// TIA Portal V19 export
FUNCTION "AUTO_SUBOUTPUT" : Void   // FC9, LAD
{ S7_Optimized_Access := 'TRUE' }
// stored: SetENOAutomatically false
BEGIN

REGION Network 1: P-202 A RO 1 FEED PUMP
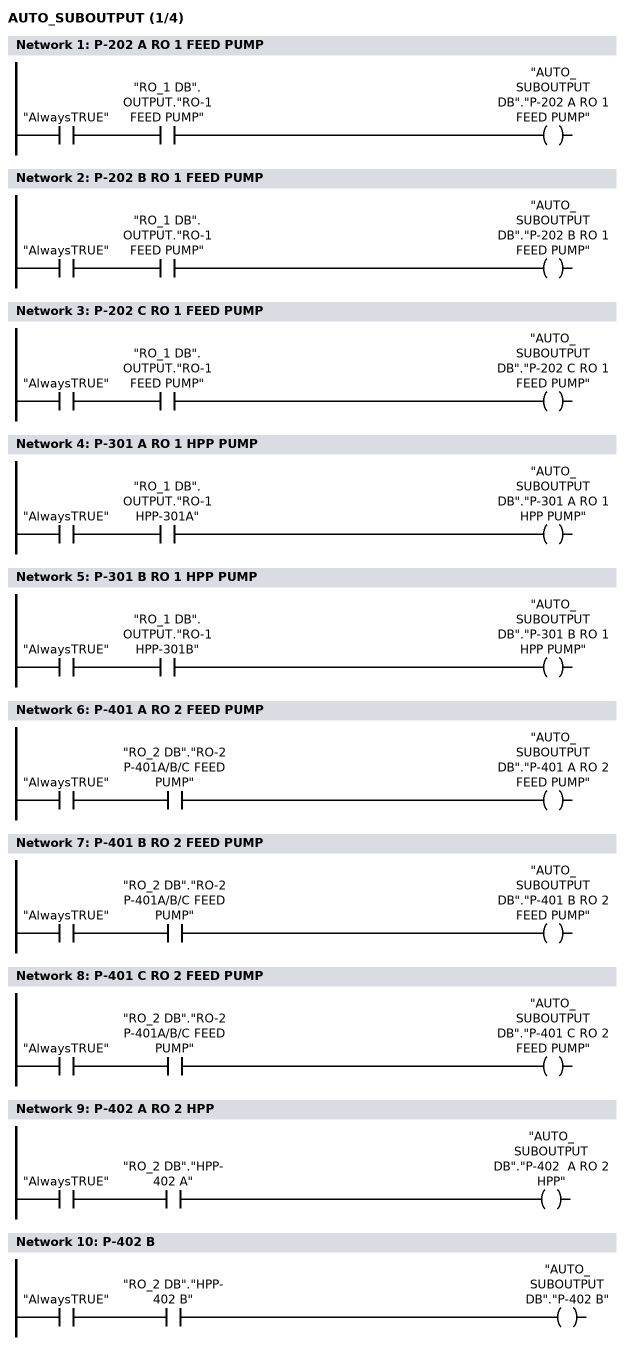
   RUNG wire#powerrail
      Contact( "AlwaysTRUE" )
      Contact( "RO_1 DB".OUTPUT."RO-1 FEED PUMP" )
      Coil( "AUTO_SUBOUTPUT DB"."P-202 A RO 1 FEED PUMP" )
   END_RUNG
   // the same network as SCL:
   "AUTO_SUBOUTPUT DB"."P-202 A RO 1 FEED PUMP" := "AlwaysTRUE" AND "RO_1 DB".OUTPUT."RO-1 FEED PUMP";
END_REGION

REGION Network 2: P-202 B RO 1 FEED PUMP
   RUNG wire#powerrail
      Contact( "AlwaysTRUE" )
      Contact( "RO_1 DB".OUTPUT."RO-1 FEED PUMP" )
      Coil( "AUTO_SUBOUTPUT DB"."P-202 B RO 1 FEED PUMP" )
   END_RUNG
   // the same network as SCL:
   "AUTO_SUBOUTPUT DB"."P-202 B RO 1 FEED PUMP" := "AlwaysTRUE" AND "RO_1 DB".OUTPUT."RO-1 FEED PUMP";
END_REGION

REGION Network 3: P-202 C RO 1 FEED PUMP
   RUNG wire#powerrail
      Contact( "AlwaysTRUE" )
      Contact( "RO_1 DB".OUTPUT."RO-1 FEED PUMP" )
      Coil( "AUTO_SUBOUTPUT DB"."P-202 C RO 1 FEED PUMP" )
   END_RUNG
   // the same network as SCL:
   "AUTO_SUBOUTPUT DB"."P-202 C RO 1 FEED PUMP" := "AlwaysTRUE" AND "RO_1 DB".OUTPUT."RO-1 FEED PUMP";
END_REGION

REGION Network 4: P-301 A RO 1 HPP PUMP
   RUNG wire#powerrail
      Contact( "AlwaysTRUE" )
      Contact( "RO_1 DB".OUTPUT."RO-1 HPP-301A" )
      Coil( "AUTO_SUBOUTPUT DB"."P-301 A RO 1 HPP PUMP" )
   END_RUNG
   // the same network as SCL:
   "AUTO_SUBOUTPUT DB"."P-301 A RO 1 HPP PUMP" := "AlwaysTRUE" AND "RO_1 DB".OUTPUT."RO-1 HPP-301A";
END_REGION

REGION Network 5: P-301 B RO 1 HPP PUMP
   RUNG wire#powerrail
      Contact( "AlwaysTRUE" )
      Contact( "RO_1 DB".OUTPUT."RO-1 HPP-301B" )
      Coil( "AUTO_SUBOUTPUT DB"."P-301 B RO 1 HPP PUMP" )
   END_RUNG
   // the same network as SCL:
   "AUTO_SUBOUTPUT DB"."P-301 B RO 1 HPP PUMP" := "AlwaysTRUE" AND "RO_1 DB".OUTPUT."RO-1 HPP-301B";
END_REGION

REGION Network 6: P-401 A RO 2 FEED PUMP
   RUNG wire#powerrail
      Contact( "AlwaysTRUE" )
      Contact( "RO_2 DB"."RO-2 P-401A/B/C FEED PUMP" )
      Coil( "AUTO_SUBOUTPUT DB"."P-401 A RO 2 FEED PUMP" )
   END_RUNG
   // the same network as SCL:
   "AUTO_SUBOUTPUT DB"."P-401 A RO 2 FEED PUMP" := "AlwaysTRUE" AND "RO_2 DB"."RO-2 P-401A/B/C FEED PUMP";
END_REGION

REGION Network 7: P-401 B RO 2 FEED PUMP
   RUNG wire#powerrail
      Contact( "AlwaysTRUE" )
      Contact( "RO_2 DB"."RO-2 P-401A/B/C FEED PUMP" )
      Coil( "AUTO_SUBOUTPUT DB"."P-401 B RO 2 FEED PUMP" )
   END_RUNG
   // the same network as SCL:
   "AUTO_SUBOUTPUT DB"."P-401 B RO 2 FEED PUMP" := "AlwaysTRUE" AND "RO_2 DB"."RO-2 P-401A/B/C FEED PUMP";
END_REGION

REGION Network 8: P-401 C RO 2 FEED PUMP
   RUNG wire#powerrail
      Contact( "AlwaysTRUE" )
      Contact( "RO_2 DB"."RO-2 P-401A/B/C FEED PUMP" )
      Coil( "AUTO_SUBOUTPUT DB"."P-401 C RO 2 FEED PUMP" )
   END_RUNG
   // the same network as SCL:
   "AUTO_SUBOUTPUT DB"."P-401 C RO 2 FEED PUMP" := "AlwaysTRUE" AND "RO_2 DB"."RO-2 P-401A/B/C FEED PUMP";
END_REGION

REGION Network 9: P-402 A RO 2 HPP
   RUNG wire#powerrail
      Contact( "AlwaysTRUE" )
      Contact( "RO_2 DB"."HPP-402 A" )
      Coil( "AUTO_SUBOUTPUT DB"."P-402  A RO 2 HPP" )
   END_RUNG
   // the same network as SCL:
   "AUTO_SUBOUTPUT DB"."P-402  A RO 2 HPP" := "AlwaysTRUE" AND "RO_2 DB"."HPP-402 A";
END_REGION

REGION Network 10: P-402 B
   RUNG wire#powerrail
      Contact( "AlwaysTRUE" )
      Contact( "RO_2 DB"."HPP-402 B" )
      Coil( "AUTO_SUBOUTPUT DB"."P-402 B" )
   END_RUNG
   // the same network as SCL:
   "AUTO_SUBOUTPUT DB"."P-402 B" := "AlwaysTRUE" AND "RO_2 DB"."HPP-402 B";
END_REGION

REGION Network 11: P-501 A EDI FEED PUMP
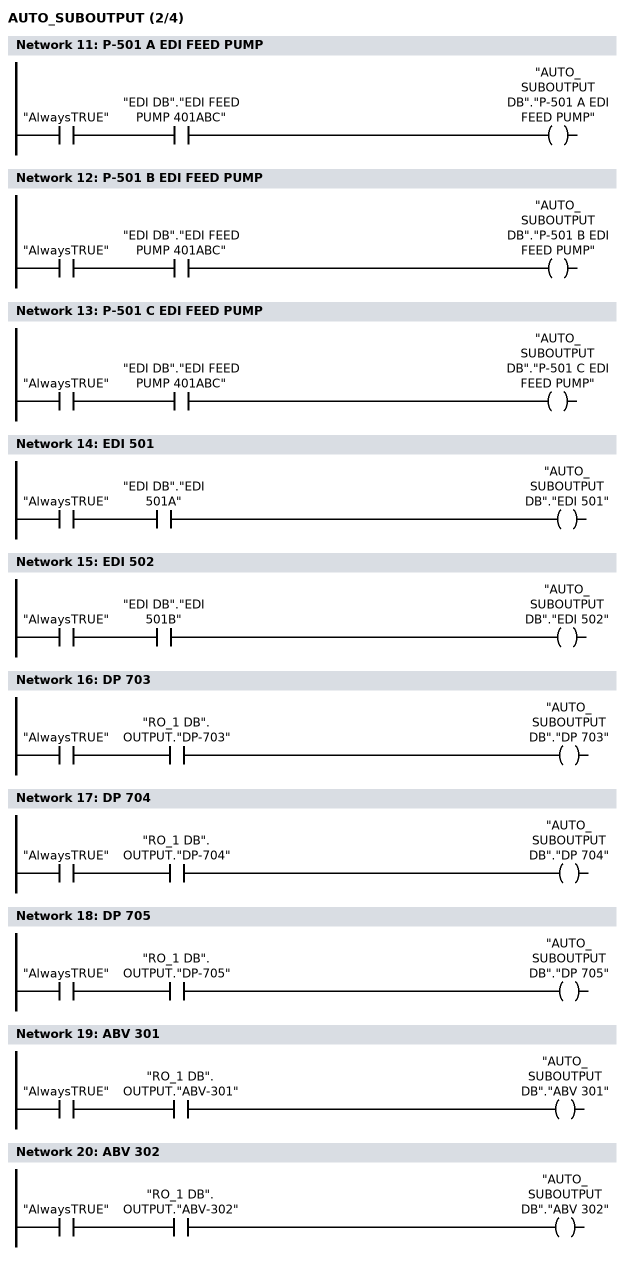
   RUNG wire#powerrail
      Contact( "AlwaysTRUE" )
      Contact( "EDI DB"."EDI FEED PUMP 401ABC" )
      Coil( "AUTO_SUBOUTPUT DB"."P-501 A EDI FEED PUMP" )
   END_RUNG
   // the same network as SCL:
   "AUTO_SUBOUTPUT DB"."P-501 A EDI FEED PUMP" := "AlwaysTRUE" AND "EDI DB"."EDI FEED PUMP 401ABC";
END_REGION

REGION Network 12: P-501 B EDI FEED PUMP
   RUNG wire#powerrail
      Contact( "AlwaysTRUE" )
      Contact( "EDI DB"."EDI FEED PUMP 401ABC" )
      Coil( "AUTO_SUBOUTPUT DB"."P-501 B EDI FEED PUMP" )
   END_RUNG
   // the same network as SCL:
   "AUTO_SUBOUTPUT DB"."P-501 B EDI FEED PUMP" := "AlwaysTRUE" AND "EDI DB"."EDI FEED PUMP 401ABC";
END_REGION

REGION Network 13: P-501 C EDI FEED PUMP
   RUNG wire#powerrail
      Contact( "AlwaysTRUE" )
      Contact( "EDI DB"."EDI FEED PUMP 401ABC" )
      Coil( "AUTO_SUBOUTPUT DB"."P-501 C EDI FEED PUMP" )
   END_RUNG
   // the same network as SCL:
   "AUTO_SUBOUTPUT DB"."P-501 C EDI FEED PUMP" := "AlwaysTRUE" AND "EDI DB"."EDI FEED PUMP 401ABC";
END_REGION

REGION Network 14: EDI 501
   RUNG wire#powerrail
      Contact( "AlwaysTRUE" )
      Contact( "EDI DB"."EDI 501A" )
      Coil( "AUTO_SUBOUTPUT DB"."EDI 501" )
   END_RUNG
   // the same network as SCL:
   "AUTO_SUBOUTPUT DB"."EDI 501" := "AlwaysTRUE" AND "EDI DB"."EDI 501A";
END_REGION

REGION Network 15: EDI 502
   RUNG wire#powerrail
      Contact( "AlwaysTRUE" )
      Contact( "EDI DB"."EDI 501B" )
      Coil( "AUTO_SUBOUTPUT DB"."EDI 502" )
   END_RUNG
   // the same network as SCL:
   "AUTO_SUBOUTPUT DB"."EDI 502" := "AlwaysTRUE" AND "EDI DB"."EDI 501B";
END_REGION

REGION Network 16: DP 703
   RUNG wire#powerrail
      Contact( "AlwaysTRUE" )
      Contact( "RO_1 DB".OUTPUT."DP-703" )
      Coil( "AUTO_SUBOUTPUT DB"."DP 703" )
   END_RUNG
   // the same network as SCL:
   "AUTO_SUBOUTPUT DB"."DP 703" := "AlwaysTRUE" AND "RO_1 DB".OUTPUT."DP-703";
END_REGION

REGION Network 17: DP 704
   RUNG wire#powerrail
      Contact( "AlwaysTRUE" )
      Contact( "RO_1 DB".OUTPUT."DP-704" )
      Coil( "AUTO_SUBOUTPUT DB"."DP 704" )
   END_RUNG
   // the same network as SCL:
   "AUTO_SUBOUTPUT DB"."DP 704" := "AlwaysTRUE" AND "RO_1 DB".OUTPUT."DP-704";
END_REGION

REGION Network 18: DP 705
   RUNG wire#powerrail
      Contact( "AlwaysTRUE" )
      Contact( "RO_1 DB".OUTPUT."DP-705" )
      Coil( "AUTO_SUBOUTPUT DB"."DP 705" )
   END_RUNG
   // the same network as SCL:
   "AUTO_SUBOUTPUT DB"."DP 705" := "AlwaysTRUE" AND "RO_1 DB".OUTPUT."DP-705";
END_REGION

REGION Network 19: ABV 301
   RUNG wire#powerrail
      Contact( "AlwaysTRUE" )
      Contact( "RO_1 DB".OUTPUT."ABV-301" )
      Coil( "AUTO_SUBOUTPUT DB"."ABV 301" )
   END_RUNG
   // the same network as SCL:
   "AUTO_SUBOUTPUT DB"."ABV 301" := "AlwaysTRUE" AND "RO_1 DB".OUTPUT."ABV-301";
END_REGION

REGION Network 20: ABV 302
   RUNG wire#powerrail
      Contact( "AlwaysTRUE" )
      Contact( "RO_1 DB".OUTPUT."ABV-302" )
      Coil( "AUTO_SUBOUTPUT DB"."ABV 302" )
   END_RUNG
   // the same network as SCL:
   "AUTO_SUBOUTPUT DB"."ABV 302" := "AlwaysTRUE" AND "RO_1 DB".OUTPUT."ABV-302";
END_REGION

REGION Network 21: AGLV-301
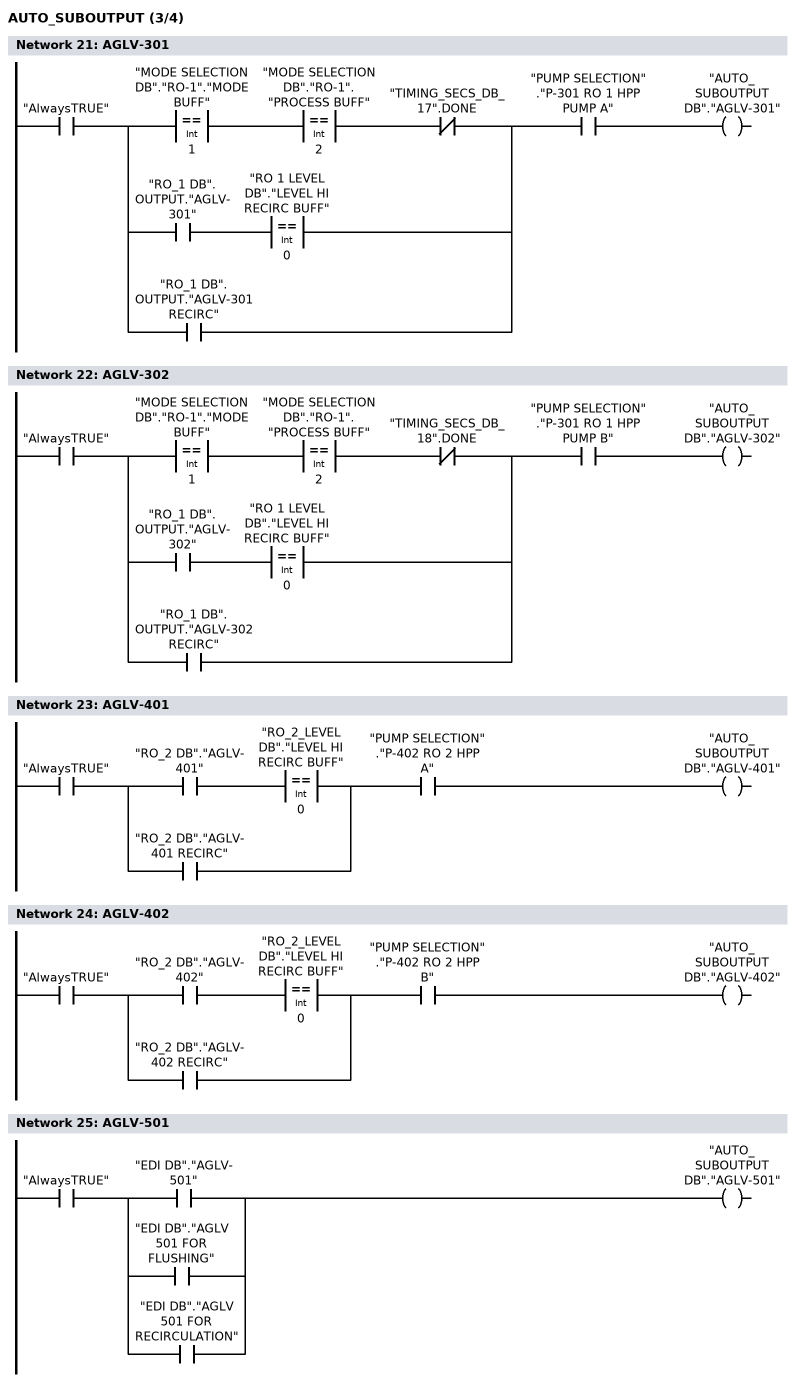
   RUNG wire#powerrail
      Contact( "AlwaysTRUE" )
      wire#w1
      { S7_Templates := "SrcType := Int" } EQ_Contact(in1 := "MODE SELECTION DB"."RO-1"."MODE BUFF", in2 := 1)
      { S7_Templates := "SrcType := Int" } EQ_Contact(in1 := "MODE SELECTION DB"."RO-1"."PROCESS BUFF", in2 := 2)
      I_Contact( "TIMING_SECS_DB_17".DONE )
      wire#w2
      Contact( "PUMP SELECTION"."P-301 RO 1 HPP PUMP A" )
      Coil( "AUTO_SUBOUTPUT DB"."AGLV-301" )
   END_RUNG
   RUNG wire#w1
      Contact( "RO_1 DB".OUTPUT."AGLV-301" )
      { S7_Templates := "SrcType := Int" } EQ_Contact(in1 := "RO 1 LEVEL DB"."LEVEL HI RECIRC BUFF", in2 := 0)
   END_RUNG wire#w2
   RUNG wire#w1
      Contact( "RO_1 DB".OUTPUT."AGLV-301 RECIRC" )
   END_RUNG wire#w2
   // the same network as SCL:
   "AUTO_SUBOUTPUT DB"."AGLV-301" := "AlwaysTRUE" AND ((("MODE SELECTION DB"."RO-1"."MODE BUFF" = 1) AND ("MODE SELECTION DB"."RO-1"."PROCESS BUFF" = 2) AND NOT "TIMING_SECS_DB_17".DONE) OR ("RO_1 DB".OUTPUT."AGLV-301" AND ("RO 1 LEVEL DB"."LEVEL HI RECIRC BUFF" = 0)) OR "RO_1 DB".OUTPUT."AGLV-301 RECIRC") AND "PUMP SELECTION"."P-301 RO 1 HPP PUMP A";
END_REGION

REGION Network 22: AGLV-302
   RUNG wire#powerrail
      Contact( "AlwaysTRUE" )
      wire#w1
      { S7_Templates := "SrcType := Int" } EQ_Contact(in1 := "MODE SELECTION DB"."RO-1"."MODE BUFF", in2 := 1)
      { S7_Templates := "SrcType := Int" } EQ_Contact(in1 := "MODE SELECTION DB"."RO-1"."PROCESS BUFF", in2 := 2)
      I_Contact( "TIMING_SECS_DB_18".DONE )
      wire#w2
      Contact( "PUMP SELECTION"."P-301 RO 1 HPP PUMP B" )
      Coil( "AUTO_SUBOUTPUT DB"."AGLV-302" )
   END_RUNG
   RUNG wire#w1
      Contact( "RO_1 DB".OUTPUT."AGLV-302" )
      { S7_Templates := "SrcType := Int" } EQ_Contact(in1 := "RO 1 LEVEL DB"."LEVEL HI RECIRC BUFF", in2 := 0)
   END_RUNG wire#w2
   RUNG wire#w1
      Contact( "RO_1 DB".OUTPUT."AGLV-302 RECIRC" )
   END_RUNG wire#w2
   // the same network as SCL:
   "AUTO_SUBOUTPUT DB"."AGLV-302" := "AlwaysTRUE" AND ((("MODE SELECTION DB"."RO-1"."MODE BUFF" = 1) AND ("MODE SELECTION DB"."RO-1"."PROCESS BUFF" = 2) AND NOT "TIMING_SECS_DB_18".DONE) OR ("RO_1 DB".OUTPUT."AGLV-302" AND ("RO 1 LEVEL DB"."LEVEL HI RECIRC BUFF" = 0)) OR "RO_1 DB".OUTPUT."AGLV-302 RECIRC") AND "PUMP SELECTION"."P-301 RO 1 HPP PUMP B";
END_REGION

REGION Network 23: AGLV-401
   RUNG wire#powerrail
      Contact( "AlwaysTRUE" )
      wire#w1
      Contact( "RO_2 DB"."AGLV-401" )
      { S7_Templates := "SrcType := Int" } EQ_Contact(in1 := "RO_2_LEVEL DB"."LEVEL HI RECIRC BUFF", in2 := 0)
      wire#w2
      Contact( "PUMP SELECTION"."P-402 RO 2 HPP A" )
      Coil( "AUTO_SUBOUTPUT DB"."AGLV-401" )
   END_RUNG
   RUNG wire#w1
      Contact( "RO_2 DB"."AGLV-401 RECIRC" )
   END_RUNG wire#w2
   // the same network as SCL:
   "AUTO_SUBOUTPUT DB"."AGLV-401" := "AlwaysTRUE" AND (("RO_2 DB"."AGLV-401" AND ("RO_2_LEVEL DB"."LEVEL HI RECIRC BUFF" = 0)) OR "RO_2 DB"."AGLV-401 RECIRC") AND "PUMP SELECTION"."P-402 RO 2 HPP A";
END_REGION

REGION Network 24: AGLV-402
   RUNG wire#powerrail
      Contact( "AlwaysTRUE" )
      wire#w1
      Contact( "RO_2 DB"."AGLV-402" )
      { S7_Templates := "SrcType := Int" } EQ_Contact(in1 := "RO_2_LEVEL DB"."LEVEL HI RECIRC BUFF", in2 := 0)
      wire#w2
      Contact( "PUMP SELECTION"."P-402 RO 2 HPP B" )
      Coil( "AUTO_SUBOUTPUT DB"."AGLV-402" )
   END_RUNG
   RUNG wire#w1
      Contact( "RO_2 DB"."AGLV-402 RECIRC" )
   END_RUNG wire#w2
   // the same network as SCL:
   "AUTO_SUBOUTPUT DB"."AGLV-402" := "AlwaysTRUE" AND (("RO_2 DB"."AGLV-402" AND ("RO_2_LEVEL DB"."LEVEL HI RECIRC BUFF" = 0)) OR "RO_2 DB"."AGLV-402 RECIRC") AND "PUMP SELECTION"."P-402 RO 2 HPP B";
END_REGION

REGION Network 25: AGLV-501
   RUNG wire#powerrail
      Contact( "AlwaysTRUE" )
      wire#w1
      Contact( "EDI DB"."AGLV-501" )
      wire#w2
      Coil( "AUTO_SUBOUTPUT DB"."AGLV-501" )
   END_RUNG
   RUNG wire#w1
      Contact( "EDI DB"."AGLV 501 FOR FLUSHING" )
   END_RUNG wire#w2
   RUNG wire#w1
      Contact( "EDI DB"."AGLV 501 FOR RECIRCULATION" )
   END_RUNG wire#w2
   // the same network as SCL:
   "AUTO_SUBOUTPUT DB"."AGLV-501" := "AlwaysTRUE" AND ("EDI DB"."AGLV-501" OR "EDI DB"."AGLV 501 FOR FLUSHING" OR "EDI DB"."AGLV 501 FOR RECIRCULATION");
END_REGION

REGION Network 26: AGLV-502
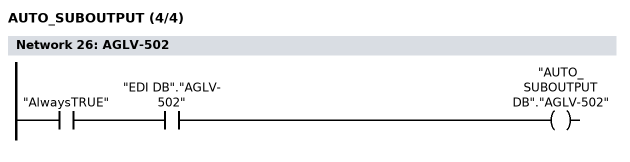
   RUNG wire#powerrail
      Contact( "AlwaysTRUE" )
      Contact( "EDI DB"."AGLV-502" )
      Coil( "AUTO_SUBOUTPUT DB"."AGLV-502" )
   END_RUNG
   // the same network as SCL:
   "AUTO_SUBOUTPUT DB"."AGLV-502" := "AlwaysTRUE" AND "EDI DB"."AGLV-502";
END_REGION
END_FUNCTION
